FUNCTION_BLOCK BrandAlarm EXTENDS FB_PIZZA_OVEN
VAR_INPUT
	
END_VAR
VAR_OUTPUT
END_VAR
VAR
END_VAR

PROPERTY BrandAlarm : BOOL
GET
BrandAlarm:=_brand_alarm;
END_GET
SET
_brand_alarm:=BrandAlarm;
END_SET
END_PROPERTY

METHOD MethodSetAlarm : BOOL
VAR_INPUT
END_VAR
IF _pizza_fertig AND _pizza_backen THEN
_brand_alarm:=TRUE;
END_IF
END_METHOD

END_FUNCTION_BLOCK

(* stored: Version 1.1.0.1, ProductVersion 3.1.4022.6
   POU BrandAlarm: Id {61dd71ff-67b5-4776-8f33-e70f3af8451a}, SpecialFunc None
   Property BrandAlarm: Id {5a7dd443-b2d8-47fa-a80f-4fef296b9646}
   Get Get: Id {68e4276e-2336-4c51-8cd5-1a5d33ac47a3}
   Set Set: Id {3723f45c-dc27-4224-87c2-e9c0ec0e40cf}
   Method MethodSetAlarm: Id {9965b012-9aa4-4715-a8d3-026a696b8cca} *)
